PROGRAM main
VAR
	Input_Switch AT %IX0.0 : bool;
	Output_Indicator AT %QX0.0 : bool;
END_VAR

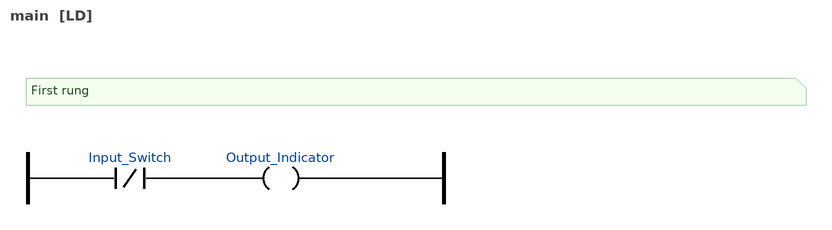
(* LD diagram, written out as Structured Text *)
(* First rung *)
Output_Indicator := NOT Input_Switch;
END_PROGRAM
